// TwinCAT 3 PLC project ExamplePLCProject
// ProgramVersion: 3.1.4023.0
// libraries:
//   Tc2_Standard, * (Beckhoff Automation GmbH)
//   Tc2_System, * (Beckhoff Automation GmbH)
//   Tc3_BA2_Common, * (Beckhoff Automation GmbH)
//   Tc3_Module, * (Beckhoff Automation GmbH)
// project tree:
//   DUTs/ ST_MonitoredAttribute.TcDUT, ST_MonitoredDevice.TcDUT, U_NumberPointer.TcDUT, U_Number.TcDUT, ST_HybridStarterControlInputBits.TcDUT, ST_HybridStarterControlOutputBits.TcDUT, U_FourByteDigitalControlInput.TcDUT, U_HybridStarterControlInput.TcDUT, U_HybridStarterControlOutput.TcDUT, U_ProfinetDeviceCtrlOutput.TcDUT, U_ProfinetDeviceDiagInput.TcDUT, U_ProfinetDeviceStateInput.TcDUT
//   GVLs/ G_Hybrid.TcGVL
//   / PlcTask.TcTTO
//   POUs/ FB_BaseDevice.TcPOU, FB_DeviceMonitor.TcPOU, FB_HybridStarter.TcPOU, FB_IOLinkDevice.TcPOU, FB_MonitoredAttribute.TcPOU, FB_MonitoredDevice.TcPOU, FB_ProfinetDevice.TcPOU, ITF_DeviceStatus.TcIO, ITF_InputDevice.TcIO, ITF_OutputDevice.TcIO, MAIN.TcPOU
// real-time tasks:
//   TASK PlcTask: cycle T#10ms, priority 20, ADS port 350

CONFIGURATION ExamplePLCProject
    RESOURCE PLC ON TwinCAT3
        TASK PlcTask(INTERVAL := T#10ms, PRIORITY := 20);
        PROGRAM MAIN WITH PlcTask : MAIN;
    END_RESOURCE
END_CONFIGURATION

// ---- DUTs/ST_MonitoredAttribute.TcDUT
TYPE ST_MonitoredAttribute :
STRUCT
	attribute : FB_MonitoredAttribute;
	attributeId : DINT;
	deviceId : DINT;
END_STRUCT
END_TYPE

// ---- DUTs/ST_MonitoredDevice.TcDUT
TYPE ST_MonitoredDevice :
STRUCT
	device : FB_MonitoredDevice;
	deviceId : DINT;
END_STRUCT
END_TYPE

// ---- DUTs/U_NumberPointer.TcDUT
// A POINTER for every data type of ANY_NUM
// PS. A pointer has the exact same size for any type
TYPE U_NumberPointer :
UNION
    // Floats
    _REAL: POINTER TO REAL;
    _LREAL: POINTER TO LREAL;
    
    // Unsigned Ints
    _USINT : POINTER TO USINT;
    _UINT  : POINTER TO UINT;
    _UDINT : POINTER TO UDINT;
    _ULINT : POINTER TO ULINT;
    
    // Signed Ints
    _SINT : POINTER TO SINT;
    _INT  : POINTER TO INT;
    _DINT : POINTER TO DINT;
    _LINT : POINTER TO LINT;
END_UNION
END_TYPE

// ---- DUTs/U_Number.TcDUT
// Every data type of ANY_NUM
TYPE U_Number :
UNION
    // Floats
    _REAL  : REAL;
    _LREAL : LREAL;
    
    // Unsigned Ints
    _USINT : USINT;
    _UINT  : UINT;
    _UDINT : UDINT;
    _ULINT : ULINT;
    
    // Signed Ints
    _SINT : SINT;
    _INT  : INT;
    _DINT : DINT;
    _LINT : LINT;
END_UNION
END_TYPE

// ---- DUTs/ST_HybridStarterControlInputBits.TcDUT
TYPE
    ST_HybridStarterControlInputBits :
    STRUCT
        Controllable              : BIT;
        ForwardRunning            : BIT;
        ReverseRunning            : BIT;
        EnableSignal              : BIT;
        Reserved4                 : BIT;
        InternalDeviceError1      : BIT;
        NominalCurrentAckExpected : BIT;
        InternalDeviceError2      : BIT;
        Reserved8                 : BIT;
        OverloadPreWarning        : BIT;
        Overload                  : BIT;
        Blocking                  : BIT;
        PhaseImbalanceGte33Lt67   : BIT;
        PhaseImbalanceGte67       : BIT;
        PhaseFailure              : BIT;
        MainsPowerFailure         : BIT;
    END_STRUCT
END_TYPE

// ---- DUTs/ST_HybridStarterControlOutputBits.TcDUT
TYPE
    ST_HybridStarterControlOutputBits :
    STRUCT
        ForwardRunning       : BIT;
        ReverseRunning       : BIT;
        ManualReset          : BIT;
        AutomaticReset       : BIT;
        Reserved4            : BIT;
        Reserved5            : BIT;
        Reserved6            : BIT;
        Reserved7            : BIT;
        NominalMotorCurrent0 : BIT;
        NominalMotorCurrent1 : BIT;
        NominalMotorCurrent2 : BIT;
        NominalMotorCurrent3 : BIT;
        Reserved12           : BIT;
        Reserved13           : BIT;
        Reserved14           : BIT;
        IdentificationValid  : BIT;
    END_STRUCT
END_TYPE

// ---- DUTs/U_FourByteDigitalControlInput.TcDUT
TYPE
    U_FourByteDigitalControlInput :
    UNION
        uUint  : UINT;
        aBytes : ARRAY[0..3] OF BYTE;
    END_UNION
END_TYPE

// ---- DUTs/U_HybridStarterControlInput.TcDUT
TYPE
    U_HybridStarterControlInput :
    UNION
        uUint  : UINT;
        aBytes : ARRAY[0..1] OF BYTE;
        stBits : ST_HybridStarterControlInputBits;
    END_UNION
END_TYPE

// ---- DUTs/U_HybridStarterControlOutput.TcDUT
TYPE
    U_HybridStarterControlOutput :
    UNION
        uUint  : UINT;
        aBytes : ARRAY[0..1] OF BYTE;
		stBits : ST_HybridStarterControlOutputBits;
    END_UNION
END_TYPE

// ---- DUTs/U_ProfinetDeviceCtrlOutput.TcDUT
TYPE
    U_ProfinetDeviceCtrlOutput :
    UNION
		uUint  : UINT;
        aBytes : ARRAY[0..1] OF BYTE;
	END_UNION
END_TYPE

// ---- DUTs/U_ProfinetDeviceDiagInput.TcDUT
TYPE
    U_ProfinetDeviceDiagInput :
    UNION
        uUint  : UINT;
        aBytes : ARRAY[0..1] OF BYTE;
    END_UNION
END_TYPE

// ---- DUTs/U_ProfinetDeviceStateInput.TcDUT
TYPE
    U_ProfinetDeviceStateInput :
    UNION
        uUint  : UINT;
        aBytes : ARRAY[0..1] OF BYTE;
    END_UNION
END_TYPE

// ---- GVLs/G_Hybrid.TcGVL
{attribute 'qualified_only'}
VAR_GLOBAL
	HS_N_AS1 : FB_HybridStarter(name := "VF01", location := "Plant", description := "VF02 on Hybrid Starter HS_N_AS1");
END_VAR

// ---- POUs/ITF_DeviceStatus.TcIO
INTERFACE ITF_DeviceStatus

PROPERTY Faults : STRING
GET
END_GET
END_PROPERTY

PROPERTY StatusOK : BOOL
GET
END_GET
END_PROPERTY

END_INTERFACE

// ---- POUs/ITF_InputDevice.TcIO
INTERFACE ITF_InputDevice

METHOD ReadControlInputs : BOOL
VAR_INPUT
END_VAR
END_METHOD

END_INTERFACE

// ---- POUs/ITF_OutputDevice.TcIO
INTERFACE ITF_OutputDevice

METHOD WriteControlOutputs : BOOL
VAR_INPUT
END_VAR
END_METHOD

END_INTERFACE

// ---- POUs/MAIN.TcPOU
PROGRAM MAIN
VAR
	bSetupDone         : BOOL;
	DeviceMonitor      : FB_DeviceMonitor;
	monitoredDevice    : FB_MonitoredDevice;
	monitoredAttribute : FB_MonitoredAttribute;
END_VAR

IF NOT bSetupDone THEN
	(*
	  Create an instance of the Phoenix Contact Hybrid Starter library - G_Hybrid.HS_N_AS1
	  This is a library that I have built
    *)
	monitoredDevice := G_Hybrid.HS_N_AS1.monitoredDevice;
	DeviceMonitor.AddMonitoredDevice(device := monitoredDevice);
	
//	// Add Current measurement TODO
//	attribute := monitoredDevice.AddMonitoredAttribute(
//		name            := "Max current",
//		inputValue      := G_Hybrid.HS_N_AS1.CurrentMaxInput,
//		monitorMaxValue := TRUE, 
//		monitorMinValue := FALSE
//	);
//	attribute.maxWarningValue._UINT := 80; // TODO set a proper value
//	attribute.maxErrorValue._UINT := 100; // TODO set a proper value
	
//	// Add Thermal load measurement TODO
//	monitoredDevice.AddMonitoredAttribute(
//		name            := "Thermal Load",
//		inputValue      := G_Hybrid.HS_N_AS1.ThermalLoadInput,
//		monitorMaxValue := TRUE,
//		monitorMinValue := FALSE
//	);
	
	bSetupDone := TRUE;
END_IF

// Read the device inputs
G_Hybrid.HS_N_AS1.ReadControlInputs();

(*
    Normal PLC code goes here
*)

// Write the control output word
G_Hybrid.HS_N_AS1.WriteControlOutput();

END_PROGRAM

// ---- POUs/FB_DeviceMonitor.TcPOU
FUNCTION_BLOCK FB_DeviceMonitor

VAR_IN_OUT
//	devices : ARRAY[*] OF FB_MonitoredDevice;
//	Devices : ARRAY[*] OF MonitoredDeviceStruct;
END_VAR

VAR
	devices : FB_BA_DynamicArray;
END_VAR

//devices.uiEntrySize := 50;

METHOD AddMonitoredDevice : BOOL // Returns the monitored device instance that has just been added
VAR_INPUT
	device : FB_MonitoredDevice;
//	name : WSTRING(255);
//	location : WSTRING(255);
//	description : WSTRING(255);
END_VAR

VAR
//	uNewMaxIndex : DINT;
//	fbMonitoredDevice : FB_MonitoredDevice;
//	stMonitoredDevice : ST_MonitoredDevice;
	resultIndex: DINT;
END_VAR
// Find the current max index in the existing array
//uNewMaxIndex := UPPER_BOUND(devices,1);

// Create a new monitored device instance
//fbMonitoredDevice.device := device.pValue;
//fbMonitoredDevice.deviceId := devices.diCount;
//device.deviceId := uNewMaxIndex;
//device.deviceId := devices.diCount;
device.deviceId := devices.LastIndex;

//fbMonitoredDevice.name := name;
//fbMonitoredDevice.location := location;
//fbMonitoredDevice.description := description;

devices.AddEntryPtr(pEntry := ADR(device));

// Populate the response struct with the instance and it's ID/index location
//stMonitoredDevice.device := fbMonitoredDevice;
//stMonitoredDevice.deviceId := uNewMaxIndex;

// Add the new device instance to the array of monitored devices
//Devices[uNewMaxIndex] := stMonitoredDevice;
//Devices[uNewMaxIndex] := fbMonitoredDevice;
//devices[uNewMaxIndex] := device;

// Return the response struct
//AddMonitoredDevice := stMonitoredDevice;
//AddMonitoredDevice := fbMonitoredDevice;
AddMonitoredDevice := TRUE;
END_METHOD

END_FUNCTION_BLOCK

// ---- POUs/FB_MonitoredDevice.TcPOU
FUNCTION_BLOCK FB_MonitoredDevice
VAR
//	Attributes : ARRAY[*] OF ST_MonitoredAttribute;
//	Attributes : ARRAY[*] OF FB_MonitoredAttribute;
//	attributes : FB_BA_DynamicArray;
END_VAR

VAR_INPUT
	// The device that is being monitored, must be a subclass of BaseDevice (i.e. `EXTENDS BaseDevice`)
//	device : POINTER TO BYTE;

	// This is the ID/index of the device in the Devices array
	deviceId : DINT;
	
	// The human-readable name of the device
	name : WSTRING(255);
	
	// The physical location in the plant
	location : WSTRING(255);
	
	description : WSTRING(255);
END_VAR

METHOD AddMonitoredAttribute : BOOL // FB_MonitoredAttribute
VAR_INPUT
	// Human-readable name
	name : WSTRING(255);

	// A loosely-typed reference to the input attribute value that needs to be monitored
	inputValue : ANY_NUM; // TODO need to consume all this in the Refresh() method

	// Determines whether or not to monitor a maximum value
	monitorMaxValue : BOOL;

	// Determines whether or not to monitor a minimum value
	monitorMinValue : BOOL;	
END_VAR

VAR
	uNewMaxIndex: DINT;
//	stMonitoredAttribute : ST_MonitoredAttribute;
//	fbMonitoredAttribute : FB_MonitoredAttribute;
END_VAR
// Find the current max index in the existing array
//uNewMaxIndex := UPPER_BOUND(Attributes,1);

// Create new monitored attributes instance
// Other variables can be set after the fact by the caller directly, on the returned instance 
//fbMonitoredAttribute.name := name;
//fbMonitoredAttribute.deviceId := deviceId;
//fbMonitoredAttribute.inputValue := inputValue;
//fbMonitoredAttribute.monitorMaxValue := monitorMaxValue;
//fbMonitoredAttribute.monitorMaxValue := monitorMaxValue;

// Populate the response struct with the instance and it's ID/index location
//stMonitoredAttribute.attribute := fbMonitoredAttribute;
//stMonitoredAttribute.attributeId := uNewMaxIndex;
//stMonitoredAttribute.deviceId := uNewMaxIndex;

// Add the new attributes instance to the array of monitored attributes
//Attributes[uNewMaxIndex] := stMonitoredAttribute;
//Attributes[uNewMaxIndex] := fbMonitoredAttribute;

// Return the response struct
//AddMonitoredDevice := stMonitoredAttribute;
//AddMonitoredAttribute := fbMonitoredAttribute;
AddMonitoredAttribute := TRUE;
END_METHOD

END_FUNCTION_BLOCK

// ---- POUs/FB_MonitoredAttribute.TcPOU
FUNCTION_BLOCK FB_MonitoredAttribute

VAR_INPUT
	// Human-readable name
	name : WSTRING(255);
	
	// Parent device ID
	deviceId : DINT;

	// A loosely-typed reference to the input attribute value that needs to be monitored
	inputValue : ANY_NUM;
	
	// Monitor the minimum value
	monitorMinValue : BOOL;

	// Min value warning threshold
	minWarningValue : U_Number;
	
	// Min value error threshold
	minErrorValue : U_Number;
	
	// Monitor the maximum value
	monitorMaxValue : BOOL;

	// Max value warning threshold
	maxWarningValue : U_Number;
	
	// Max value error threshold
	maxErrorValue : U_Number;
	
	// Initial grace period - default 2 seconds
	initialGracePeriod : TIME := T#2S;
	
	// Use the override value below (provided by the Operator)
	useOverrideValue : BOOL;

	// Manually override the value for simulation etc
	overrideValue : ANY_NUM;
	
	// Skip any warnings if set to TRUE
	skipWarnings : BOOL;

	// Skip any errors if set to TRUE
	skipErrors : BOOL;
	
END_VAR

VAR_OUTPUT
	// A pointer to the current value of the monitored attribute - kept updated by the Refresh() method
	currentValuePointer : U_Number;
END_VAR

VAR
	// A const to determine the type
	valueType : STRING(8);
END_VAR

METHOD Refresh : BOOL

VAR
	uNumPointer : U_NumberPointer;
END_VAR
CASE inputValue.TypeClass OF
        __SYSTEM.TYPE_CLASS.TYPE_REAL:
                uNumPointer._REAL := inputValue.pValue;
                currentValuePointer._REAL := uNumPointer._REAL^;
                valueType := 'REAL';
        __SYSTEM.TYPE_CLASS.TYPE_LREAL:
                uNumPointer._LREAL := inputValue.pValue;
                currentValuePointer._LREAL := uNumPointer._LREAL^;
                valueType := 'LREAL';
        __SYSTEM.TYPE_CLASS.TYPE_USINT:
                uNumPointer._USINT := inputValue.pValue;
                currentValuePointer._USINT := uNumPointer._USINT^;
                valueType := 'USINT';
        __SYSTEM.TYPE_CLASS.TYPE_UINT:
                uNumPointer._UINT := inputValue.pValue;
                currentValuePointer._UINT := uNumPointer._UINT^;
                valueType := 'UINT';
        __SYSTEM.TYPE_CLASS.TYPE_UDINT:
                uNumPointer._UDINT := inputValue.pValue;
                currentValuePointer._UDINT := uNumPointer._UDINT^;
                valueType := 'UDINT';
        __SYSTEM.TYPE_CLASS.TYPE_ULINT:
                uNumPointer._ULINT := inputValue.pValue;
                currentValuePointer._ULINT := uNumPointer._ULINT^;
                valueType := 'ULINT';
        __SYSTEM.TYPE_CLASS.TYPE_SINT:
                uNumPointer._SINT := inputValue.pValue;
                currentValuePointer._SINT := uNumPointer._SINT^;
                valueType := 'SINT';
        __SYSTEM.TYPE_CLASS.TYPE_INT:
                uNumPointer._INT := inputValue.pValue;
                currentValuePointer._INT := uNumPointer._INT^;
                valueType := 'INT';
        __SYSTEM.TYPE_CLASS.TYPE_DINT:
                uNumPointer._DINT := inputValue.pValue;
                currentValuePointer._DINT := uNumPointer._DINT^;
                valueType := 'DINT';
        __SYSTEM.TYPE_CLASS.TYPE_LINT:
                uNumPointer._LINT := inputValue.pValue;
                currentValuePointer._LINT := uNumPointer._LINT^;
                valueType := 'LINT';

ELSE
        currentValuePointer._INT := 0;
END_CASE;
END_METHOD

END_FUNCTION_BLOCK

// ---- POUs/FB_HybridStarter.TcPOU
FUNCTION_BLOCK FB_HybridStarter EXTENDS FB_BaseDevice
VAR_INPUT
	// The control output to the starter
    ControlOutput    AT %Q* : UINT;
	// The 5in1 state data word from the starter
    StatusInput      AT %I* : UINT;
	// The Max. current ampere word from the starter, in 10s of mA
    CurrentMaxInput  AT %I* : UINT;
	// The Thermal load input word from the starter
    ThermalLoadInput AT %I* : UINT;

    // Local copy of main control word as UINT (same as ControlOutput)
    uControl : UINT;
    // Local copy of main control word, individual bits that are translated to send to output
    stControl : ST_HybridStarterControlOutputBits;

    // Local copy of main status word as UINT (same as StatusInput)
    uStatus : UINT;
    // Local copy of main status word, translated to be readable as individual bits
    stStatus : ST_HybridStarterControlInputBits;

    // Max current word, multiplied by 10x, from tens of mA (same as CurrentMaxInput) to hundreds of mA, to be human readable
    uCurrentMilliamps : UINT;

    // Motor thermal load percentage (same as ThermalLoadInput)
    uThermalLoadPercent : UINT;
END_VAR

VAR
    uControlOutput : U_HybridStarterControlOutput;
    uControlInput1 : U_HybridStarterControlInput;
END_VAR

METHOD ReadControlInputs : BOOL
uStatus             := StatusInput;
uCurrentMilliamps   := CurrentMaxInput * 10; // Turn the 10s of mA value into 100s of mA
uThermalLoadPercent := ThermalLoadInput;

// Run the main input UINT through the union and store the bits in the local struct VAR
uControlInput1.uUint := uStatus;
stStatus             := uControlInput1.stBits;

ReadControlInputs := TRUE;
END_METHOD

METHOD RunForward : BOOL
VAR_INPUT
END_VAR
stControl.ForwardRunning := TRUE;
stControl.ReverseRunning := FALSE;
RunForward := TRUE;
END_METHOD

METHOD RunReverse : BOOL
VAR_INPUT
END_VAR
stControl.ForwardRunning := FALSE;
stControl.ReverseRunning := TRUE;
RunReverse := TRUE;
END_METHOD

METHOD SetNominalCurrent : BOOL
VAR_INPUT
	bit0 : BOOL;
	bit1 : BOOL;
	bit2 : BOOL;
	bit3 : BOOL;
END_VAR
stControl.NominalMotorCurrent0 := bit0;
stControl.NominalMotorCurrent1 := bit1;
stControl.NominalMotorCurrent2 := bit2;
stControl.NominalMotorCurrent3 := bit3;
stControl.IdentificationValid := TRUE;
SetNominalCurrent := TRUE;
END_METHOD

METHOD Stop : BOOL
VAR_INPUT
END_VAR
stControl.ForwardRunning := FALSE;
stControl.ReverseRunning := FALSE;

uControlOutput.stBits := stControl;
uControl := uControlOutput.uUint;
ControlOutput := uControl;

Stop := TRUE;
END_METHOD

METHOD WriteControlOutput : BOOL
VAR_INPUT
END_VAR
uControlOutput.stBits := stControl;
uControl := uControlOutput.uUint;
ControlOutput := uControl;
WriteControlOutput := TRUE;
END_METHOD

END_FUNCTION_BLOCK

// ---- POUs/FB_BaseDevice.TcPOU
FUNCTION_BLOCK ABSTRACT FB_BaseDevice

VAR_INPUT
	name : WSTRING(255);
	location : WSTRING(255);
	description : WSTRING(255);
END_VAR

VAR
	monitoredDevice : FB_MonitoredDevice;
END_VAR

monitoredDevice.name := name;
monitoredDevice.location := location;
monitoredDevice.description := description;

METHOD FB_init : BOOL
VAR_INPUT
	bInitRetains : BOOL; // if TRUE, the retain variables are initialized (warm start / cold start)
	bInCopyCode : BOOL;  // if TRUE, the instance afterwards gets moved into the copy code (online change)
	name : WSTRING(255);
	location : WSTRING(255);
	description : WSTRING(255);
END_VAR
END_METHOD

END_FUNCTION_BLOCK

// ---- POUs/FB_IOLinkDevice.TcPOU
FUNCTION_BLOCK ABSTRACT FB_IOLinkDevice EXTENDS FB_BaseDevice
VAR_INPUT
    // This is presented as a linkable input in the main project via a GVL	
    PQIStatusInput AT %I* : BYTE;
END_VAR

END_FUNCTION_BLOCK

// ---- POUs/FB_ProfinetDevice.TcPOU
FUNCTION_BLOCK ABSTRACT FB_ProfinetDevice EXTENDS FB_BaseDevice
VAR_INPUT
    // This is presented as a linkable input in the main project via a GVL
    StateInput AT %I* : UINT;
    // This is presented as a linkable input in the main project via a GVL
    DiagInput AT %I* : UINT;
	// This is presented as a linkable output in the main project via a GVL	
    CtrlOutput AT %Q* : UINT;
END_VAR
VAR
    uCtrlOutput : U_ProfinetDeviceCtrlOutput;
    uDiagInput  : U_ProfinetDeviceDiagInput;
    uStateInput : U_ProfinetDeviceStateInput;
END_VAR

END_FUNCTION_BLOCK
